// Mitsubishi GX Works2 project: 23   PLC: FX3G

// task Task_01 (event TRUE, interval 0, priority 31): POU_01

PROGRAM POU_01
VAR
  ton1 : TON;
  gas : INT;
END_VAR
IF M8002 THEN
	gas := 0;
END_IF;
IF NOT M1 THEN
	gas:=0;
END_IF;

CASE gas OF
0:
Y0:=FALSE;
Y1:=FALSE;
Y2:=FALSE;
Y3:=FALSE;
IF M1=TRUE THEN
	gas:=1;
END_IF;

1:
Y0:=TRUE;
Y1:=TRUE;
ton1(IN := NOT ton1.Q, PT := T#5s);
IF ton1.Q THEN
	gas:=2;
END_IF;
	
2:	
Y2:=TRUE;
ton1(IN := NOT ton1.Q, PT := T#10s);
IF ton1.Q THEN
	Y3:=TRUE;
END_IF;

END_CASE;
END_PROGRAM
